(* PLC project Trafik_Lambasi_Yaya.project, CODESYS CODESYS V3.5 SP21 Patch 5 *)
(* stored: creationDateTime 2026-07-28T18:28:46.7939622, modificationDateTime 2026-07-28T18:26:22.4681049 *)

PROGRAM PLC_PRG
  VAR
    start : BOOL;
    Stop : BOOL;
    sistem_aktif : BOOL;
    T1 : TON;
    kirmizi : BOOL;
    sari : BOOL;
    yesil : BOOL;
    sari_kosul2 : BOOL;
    sari_gercek : BOOL;
    sari_kosul1 : BOOL;
    yaya_yesil : BOOL;
    yaya_kirmizi : BOOL;
    yaya_buton : BOOL;
    yaya_istek : BOOL;
    T2 : TON;
  END_VAR
  VAR  (* added by the conversion: wires and edge detectors of the diagram *)
    _LE16_ENO : BOOL;
    _LE16_OUT : BOOL;
    _GE25_ENO : BOOL;
    _GE25_OUT : BOOL;
    _LE24_ENO : BOOL;
    _LE24_OUT : BOOL;
    _GE32_ENO : BOOL;
    _GE32_OUT : BOOL;
    _LE31_ENO : BOOL;
    _LE31_OUT : BOOL;
    _GE46_ENO : BOOL;
    _GE46_OUT : BOOL;
    _LE45_ENO : BOOL;
    _LE45_OUT : BOOL;
  END_VAR

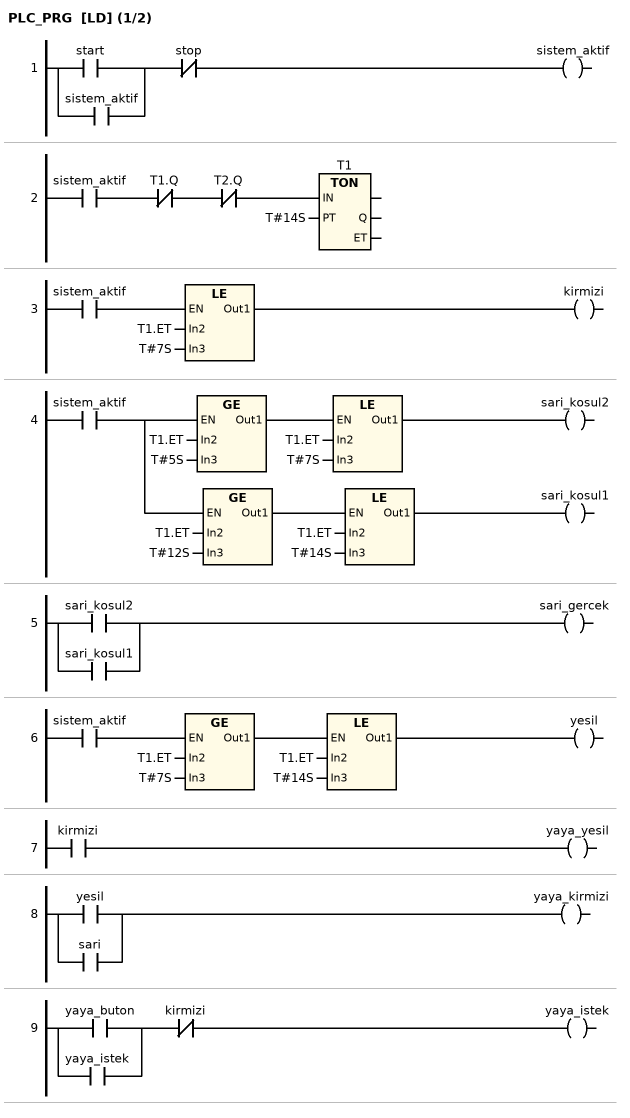
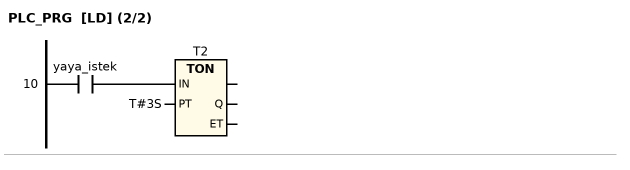
(* LD diagram, written out as Structured Text *)

sistem_aktif := (start OR sistem_aktif) AND NOT stop;

T1(IN := sistem_aktif AND NOT T1.Q AND NOT T2.Q, PT := T#14S);

_LE16_OUT := LE(EN := sistem_aktif, IN1 := T1.ET, IN2 := T#7S, ENO => _LE16_ENO);
kirmizi := _LE16_OUT;

_GE25_OUT := GE(EN := sistem_aktif, IN1 := T1.ET, IN2 := T#5S, ENO => _GE25_ENO);
_LE24_OUT := LE(EN := _GE25_OUT, IN1 := T1.ET, IN2 := T#7S, ENO => _LE24_ENO);
sari_kosul2 := _LE24_OUT;
_GE32_OUT := GE(EN := sistem_aktif, IN1 := T1.ET, IN2 := T#12S, ENO => _GE32_ENO);
_LE31_OUT := LE(EN := _GE32_OUT, IN1 := T1.ET, IN2 := T#14S, ENO => _LE31_ENO);
sari_kosul1 := _LE31_OUT;

sari_gercek := sari_kosul2 OR sari_kosul1;

_GE46_OUT := GE(EN := sistem_aktif, IN1 := T1.ET, IN2 := T#7S, ENO => _GE46_ENO);
_LE45_OUT := LE(EN := _GE46_OUT, IN1 := T1.ET, IN2 := T#14S, ENO => _LE45_ENO);
yesil := _LE45_OUT;

yaya_yesil := kirmizi;

yaya_kirmizi := yesil OR sari;

yaya_istek := (yaya_buton OR yaya_istek) AND NOT kirmizi;

T2(IN := yaya_istek, PT := T#3S);
END_PROGRAM
